TYPE RemoteFeedbackMru :
STRUCT

END_STRUCT
END_TYPE

(* stored: Version 1.1.0.1, ProductVersion 3.1.4020.12
   DUT RemoteFeedbackMru: Id {e5da7f68-9b82-4c49-ac9c-e08f2e5a864f} *)
